DATA_BLOCK "ST10_Flow27_KReserveLoad&Unload_iDB"
{ S7_Optimized_Access := 'TRUE' }
VERSION : 0.1
NON_RETAIN
// ATTRIBUTES
// AUTO_NUMBER = False
// BLOCK_NUMBER = 1097
// END_ATTRIBUTES
"ST10_Flow27_KReserveLoad&Unload"

BEGIN

END_DATA_BLOCK

